LIN {X 0,Y 114.928,Z 408.229,A -85,B 0,C 180,E1 -30802.349,E2 -30802.349} C_VEL
LIN {X 0,Y 112.852,Z 415.99,A -85,B 0,C 180,E1 -30806.603,E2 -30806.603} C_VEL
LIN {X 0,Y 110.875,Z 424.848,A -85,B 0,C 180,E1 -30812.549,E2 -30812.549} C_VEL
LIN {X 0,Y 109.952,Z 432.134,A -85,B 0,C 180,E1 -30818.427,E2 -30818.427} C_VEL
LIN {X 0,Y 110.137,Z 438.588,A -85,B 0,C 180,E1 -30824.579,E2 -30824.579} C_VEL
LIN {X 0,Y 111.737,Z 444.355,A -85,B 0,C 180,E1 -30831.025,E2 -30831.025} C_VEL
LIN {X 0,Y 115.537,Z 449.975,A -85,B 0,C 180,E1 -30838.383,E2 -30838.383} C_VEL
LIN {X 0,Y 120.475,Z 454.059,A -85,B 0,C 180,E1 -30844.487,E2 -30844.487} C_VEL
LIN {X 0,Y 127.737,Z 457.673,A -85,B 0,C 180,E1 -30850.724,E2 -30850.724} C_VEL
LIN {X 0,Y 137.278,Z 460.508,A -85,B 0,C 180,E1 -30856.577,E2 -30856.577} C_VEL
LIN {X 0,Y 149.17,Z 462.456,A -85,B 0,C 180,E1 -30861.875,E2 -30861.875} C_VEL
LIN {X 0,Y 161.996,Z 463.408,A -85,B 0,C 180,E1 -30866.197,E2 -30866.197} C_VEL
LIN {X 0,Y 172.889,Z 463.546,A -85,B 0,C 180,E1 -30869.172,E2 -30869.172} C_VEL
LIN {X 0,Y 171.419,Z 463.614,A -85,B 0,C 180,E1 -30869.286,E2 -30869.286} C_VEL
LIN {X 0,Y 166.186,Z 463.751,A -85,B 0,C 180,E1 -30868.796,E2 -30868.796} C_VEL
LIN {X 0,Y 154.259,Z 463.825,A -85,B 0,C 180,E1 -30866.675,E2 -30866.675} C_VEL
LIN {X 0,Y 146.999,Z 463.619,A -85,B 0,C 180,E1 -30864.785,E2 -30864.785} C_VEL
LIN {X 0,Y 144.8,Z 463.468,A -85,B 0,C 180,E1 -30864.025,E2 -30864.025} C_VEL
LIN {X 0,Y 129.691,Z 461.525,A -85,B 0,C 180,E1 -30857.262,E2 -30857.262} C_VEL
LIN {X 0,Y 123.495,Z 460.082,A -85,B 0,C 180,E1 -30853.468,E2 -30853.468} C_VEL
LIN {X 0,Y 114.996,Z 456.746,A -85,B 0,C 180,E1 -30846.448,E2 -30846.448} C_VEL
LIN {X 0,Y 108.181,Z 451.593,A -85,B 0,C 180,E1 -30837.619,E2 -30837.619} C_VEL
LIN {X 0,Y 105.024,Z 446.619,A -85,B 0,C 180,E1 -30830.311,E2 -30830.311} C_VEL
LIN {X 0,Y 103.823,Z 441.564,A -85,B 0,C 180,E1 -30823.894,E2 -30823.894} C_VEL
LIN {X 0,Y 104.011,Z 435.561,A -85,B 0,C 180,E1 -30817.451,E2 -30817.451} C_VEL
LIN {X 0,Y 105.361,Z 428.686,A -85,B 0,C 180,E1 -30811.268,E2 -30811.268} C_VEL
LIN {X 0,Y 107.859,Z 420.234,A -85,B 0,C 180,E1 -30805.054,E2 -30805.054} C_VEL
LIN {X 0,Y 110.868,Z 411.549,A -85,B 0,C 180,E1 -30799.917,E2 -30799.917} C_VEL
LIN {X 0,Y 113.638,Z 403.688,A -85,B 0,C 180,E1 -30796.061,E2 -30796.061} C_VEL
LIN {X 0,Y 115.913,Z 396.746,A -85,B 0,C 180,E1 -30792.908,E2 -30792.908} C_VEL
LIN {X 0,Y 116.822,Z 392.502,A -85,B 0,C 180,E1 -30790.396,E2 -30790.396} C_VEL
LIN {X 0,Y 117.379,Z 389.446,A -85,B 0,C 180,E1 -30787.772,E2 -30787.772} C_VEL
LIN {X 0,Y 117.764,Z 386.797,A -85,B 0,C 180,E1 -30784.354,E2 -30784.354} C_VEL
LIN {X 0,Y 118.148,Z 384.921,A -85,B 0,C 180,E1 -30779.998,E2 -30779.998} C_VEL
LIN {X 0,Y 117.859,Z 385.788,A -85,B 0,C 180,E1 -30779.68,E2 -30779.68} C_VEL
LIN {X 0,Y 112.453,Z 398.556,A -85,B 0,C 180,E1 -30779.412,E2 -30779.412} C_VEL
LIN {X 0,Y 106.312,Z 409.458,A -85,B 0,C 180,E1 -30779.084,E2 -30779.084} C_VEL
LIN {X 0,Y 100.174,Z 418.396,A -85,B 0,C 180,E1 -30778.714,E2 -30778.714} C_VEL
LIN {X 0,Y 93.168,Z 426.917,A -85,B 0,C 180,E1 -30778.175,E2 -30778.175} C_VEL
LIN {X 0,Y 86.17,Z 434.129,A -85,B 0,C 180,E1 -30777.574,E2 -30777.574} C_VEL
LIN {X 0,Y 79.187,Z 440.326,A -85,B 0,C 180,E1 -30776.819,E2 -30776.819} C_VEL
LIN {X 0,Y 70.482,Z 446.858,A -85,B 0,C 180,E1 -30775.661,E2 -30775.661} C_VEL
LIN {X 0,Y 63.552,Z 451.36,A -85,B 0,C 180,E1 -30774.431,E2 -30774.431} C_VEL
LIN {X 0,Y 52.249,Z 457.3,A -85,B 0,C 180,E1 -30771.68,E2 -30771.68} C_VEL
LIN {X 0,Y 43.037,Z 461.18,A -85,B 0,C 180,E1 -30768.466,E2 -30768.466} C_VEL
LIN {X 0,Y 36.38,Z 463.552,A -85,B 0,C 180,E1 -30764.995,E2 -30764.995} C_VEL
LIN {X 0,Y 29.88,Z 465.354,A -85,B 0,C 180,E1 -30760.192,E2 -30760.192} C_VEL
LIN {X 0,Y 18.299,Z 467.822,A -85,B 0,C 180,E1 -30740.185,E2 -30740.185} C_VEL
LIN {X 0,Y 14.211,Z 468.422,A -85,B 0,C 180,E1 -30719.639,E2 -30719.639} C_VEL
LIN {X 0,Y 12.863,Z 468.588,A -85,B 0,C 180,E1 -30690,E2 -30690} C_VEL
LIN {X 0,Y 14.256,Z 468.423,A -85,B 0,C 180,E1 -30660.462,E2 -30660.462} C_VEL
LIN {X 0,Y 18.308,Z 467.822,A -85,B 0,C 180,E1 -30639.849,E2 -30639.849} C_VEL
LIN {X 0,Y 29.882,Z 465.355,A -85,B 0,C 180,E1 -30619.819,E2 -30619.819} C_VEL
LIN {X 0,Y 39.699,Z 462.4,A -85,B 0,C 180,E1 -30613.177,E2 -30613.177} C_VEL
LIN {X 0,Y 49.826,Z 458.409,A -85,B 0,C 180,E1 -30609.123,E2 -30609.123} C_VEL
LIN {X 0,Y 57.014,Z 455,A -85,B 0,C 180,E1 -30607.085,E2 -30607.085} C_VEL
LIN {X 0,Y 67.011,Z 449.169,A -85,B 0,C 180,E1 -30604.906,E2 -30604.906} C_VEL
LIN {X 0,Y 75.699,Z 443.075,A -85,B 0,C 180,E1 -30603.587,E2 -30603.587} C_VEL
LIN {X 0,Y 82.676,Z 437.38,A -85,B 0,C 180,E1 -30602.781,E2 -30602.781} C_VEL
LIN {X 0,Y 91.416,Z 428.834,A -85,B 0,C 180,E1 -30601.94,E2 -30601.94} C_VEL
LIN {X 0,Y 98.421,Z 420.663,A -85,B 0,C 180,E1 -30601.41,E2 -30601.41} C_VEL
LIN {X 0,Y 104.557,Z 412.158,A -85,B 0,C 180,E1 -30601.01,E2 -30601.01} C_VEL
LIN {X 0,Y 109.821,Z 403.45,A -85,B 0,C 180,E1 -30600.722,E2 -30600.722} C_VEL
LIN {X 0,Y 114.579,Z 393.859,A -85,B 0,C 180,E1 -30600.513,E2 -30600.513} C_VEL
LIN {X 0,Y 117.859,Z 385.789,A -85,B 0,C 180,E1 -30600.319,E2 -30600.319} C_VEL
LIN {X 0,Y 118.147,Z 384.922,A -85,B 0,C 180,E1 -30600.002,E2 -30600.002} C_VEL
LIN {X 0,Y 117.762,Z 386.791,A -85,B 0,C 180,E1 -30595.671,E2 -30595.671} C_VEL
LIN {X 0,Y 117.552,Z 388.558,A -85,B 0,C 180,E1 -30593.134,E2 -30593.134} C_VEL
LIN {X 0,Y 117.059,Z 391.295,A -85,B 0,C 180,E1 -30590.499,E2 -30590.499} C_VEL
LIN {X 0,Y 116.143,Z 395.768,A -85,B 0,C 180,E1 -30587.597,E2 -30587.597} C_VEL
LIN {X 0,Y 114.614,Z 400.732,A -85,B 0,C 180,E1 -30585.237,E2 -30585.237} C_VEL
LIN {X 0,Y 111.495,Z 409.774,A -85,B 0,C 180,E1 -30580.998,E2 -30580.998} C_VEL
LIN {X 0,Y 109.117,Z 416.554,A -85,B 0,C 180,E1 -30577.269,E2 -30577.269} C_VEL
LIN {X 0,Y 106.354,Z 425.079,A -85,B 0,C 180,E1 -30571.506,E2 -30571.506} C_VEL
LIN {X 0,Y 104.496,Z 432.383,A -85,B 0,C 180,E1 -30565.518,E2 -30565.518} C_VEL
LIN {X 0,Y 103.733,Z 438.549,A -85,B 0,C 180,E1 -30559.47,E2 -30559.47} C_VEL
LIN {X 0,Y 104.353,Z 444.734,A -85,B 0,C 180,E1 -30552.201,E2 -30552.201} C_VEL
LIN {X 0,Y 106.92,Z 450.051,A -85,B 0,C 180,E1 -30544.758,E2 -30544.758} C_VEL
LIN {X 0,Y 111.236,Z 454.337,A -85,B 0,C 180,E1 -30537.811,E2 -30537.811} C_VEL
LIN {X 0,Y 117.729,Z 457.962,A -85,B 0,C 180,E1 -30530.988,E2 -30530.988} C_VEL
LIN {X 0,Y 124.297,Z 460.268,A -85,B 0,C 180,E1 -30526.017,E2 -30526.017} C_VEL
LIN {X 0,Y 135.507,Z 462.502,A -85,B 0,C 180,E1 -30519.804,E2 -30519.804} C_VEL
LIN {X 0,Y 148.1,Z 463.65,A -85,B 0,C 180,E1 -30514.785,E2 -30514.785} C_VEL
LIN {X 0,Y 164.307,Z 463.8,A -85,B 0,C 180,E1 -30510,E2 -30510} C_VEL
LIN {X 0,Y 148.1,Z 463.65,A -85,B 0,C 180,E1 -30505.215,E2 -30505.215} C_VEL
LIN {X 0,Y 144.8,Z 463.468,A -85,B 0,C 180,E1 -30504.025,E2 -30504.025} C_VEL
LIN {X 0,Y 140.14,Z 463.214,A -85,B 0,C 180,E1 -30502.568,E2 -30502.568} C_VEL
LIN {X 0,Y 124.745,Z 462.622,A -85,B 0,C 180,E1 -30498.671,E2 -30498.671} C_VEL
LIN {X 0,Y 120.314,Z 462.099,A -85,B 0,C 180,E1 -30496.874,E2 -30496.874} C_VEL
LIN {X 0,Y 119.067,Z 461.847,A -85,B 0,C 180,E1 -30496.159,E2 -30496.159} C_VEL
LIN {X 0,Y 111.725,Z 459.856,A -85,B 0,C 180,E1 -30490.653,E2 -30490.653} C_VEL
LIN {X 0,Y 103.714,Z 455.76,A -85,B 0,C 180,E1 -30481.749,E2 -30481.749} C_VEL
LIN {X 0,Y 99.573,Z 451.39,A -85,B 0,C 180,E1 -30473.76,E2 -30473.76} C_VEL
LIN {X 0,Y 97.648,Z 446.43,A -85,B 0,C 180,E1 -30466.028,E2 -30466.028} C_VEL
LIN {X 0,Y 97.754,Z 439.952,A -85,B 0,C 180,E1 -30457.736,E2 -30457.736} C_VEL
LIN {X 0,Y 99.087,Z 434.239,A -85,B 0,C 180,E1 -30451.665,E2 -30451.665} C_VEL
LIN {X 0,Y 101.522,Z 427.548,A -85,B 0,C 180,E1 -30445.851,E2 -30445.851} C_VEL
LIN {X 0,Y 104.836,Z 419.615,A -85,B 0,C 180,E1 -30440.194,E2 -30440.194} C_VEL
LIN {X 0,Y 108.197,Z 411.955,A -85,B 0,C 180,E1 -30435.778,E2 -30435.778} C_VEL
LIN {X 0,Y 111.818,Z 403.365,A -85,B 0,C 180,E1 -30431.671,E2 -30431.671} C_VEL
LIN {X 0,Y 113.211,Z 399.616,A -85,B 0,C 180,E1 -30429.742,E2 -30429.742} C_VEL
LIN {X 0,Y 114.351,Z 395.944,A -85,B 0,C 180,E1 -30427.059,E2 -30427.059} C_VEL
LIN {X 0,Y 114.72,Z 394.322,A -85,B 0,C 180,E1 -30425.271,E2 -30425.271} C_VEL
LIN {X 0,Y 115.013,Z 393.127,A -85,B 0,C 180,E1 -30423.501,E2 -30423.501} C_VEL
LIN {X 0,Y 114.162,Z 394.978,A -85,B 0,C 180,E1 -30423.048,E2 -30423.048} C_VEL
LIN {X 0,Y 108.193,Z 406.5,A -85,B 0,C 180,E1 -30422.897,E2 -30422.897} C_VEL
LIN {X 0,Y 101.148,Z 417.069,A -85,B 0,C 180,E1 -30422.801,E2 -30422.801} C_VEL
LIN {X 0,Y 94.977,Z 424.806,A -85,B 0,C 180,E1 -30422.624,E2 -30422.624} C_VEL
LIN {X 0,Y 86.162,Z 433.936,A -85,B 0,C 180,E1 -30422.306,E2 -30422.306} C_VEL
LIN {X 0,Y 79.112,Z 440.133,A -85,B 0,C 180,E1 -30421.978,E2 -30421.978} C_VEL
LIN {X 0,Y 70.302,Z 446.665,A -85,B 0,C 180,E1 -30421.456,E2 -30421.456} C_VEL
LIN {X 0,Y 63.259,Z 451.165,A -85,B 0,C 180,E1 -30420.888,E2 -30420.888} C_VEL
LIN {X 0,Y 53.213,Z 456.436,A -85,B 0,C 180,E1 -30419.749,E2 -30419.749} C_VEL
LIN {X 0,Y 42.194,Z 460.986,A -85,B 0,C 180,E1 -30417.99,E2 -30417.99} C_VEL
LIN {X 0,Y 35.215,Z 463.358,A -85,B 0,C 180,E1 -30416.255,E2 -30416.255} C_VEL
LIN {X 0,Y 28.272,Z 465.161,A -85,B 0,C 180,E1 -30413.903,E2 -30413.903} C_VEL
LIN {X 0,Y 14.786,Z 467.628,A -85,B 0,C 180,E1 -30401.916,E2 -30401.916} C_VEL
LIN {X 0,Y 8.773,Z 468.229,A -85,B 0,C 180,E1 -30383.237,E2 -30383.237} C_VEL
LIN {X 0,Y 5.75,Z 468.395,A -85,B 0,C 180,E1 -30330,E2 -30330} C_VEL
LIN {X 0,Y 8.798,Z 468.23,A -85,B 0,C 180,E1 -30276.98,E2 -30276.98} C_VEL
LIN {X 0,Y 14.79,Z 467.629,A -85,B 0,C 180,E1 -30258.131,E2 -30258.131} C_VEL
LIN {X 0,Y 28.272,Z 465.161,A -85,B 0,C 180,E1 -30246.108,E2 -30246.108} C_VEL
LIN {X 0,Y 38.701,Z 462.206,A -85,B 0,C 180,E1 -30242.827,E2 -30242.827} C_VEL
LIN {X 0,Y 49.202,Z 458.215,A -85,B 0,C 180,E1 -30240.887,E2 -30240.887} C_VEL
LIN {X 0,Y 56.224,Z 455,A -85,B 0,C 180,E1 -30239.944,E2 -30239.944} C_VEL
LIN {X 0,Y 66.78,Z 448.975,A -85,B 0,C 180,E1 -30238.809,E2 -30238.809} C_VEL
LIN {X 0,Y 75.588,Z 442.882,A -85,B 0,C 180,E1 -30238.188,E2 -30238.188} C_VEL
LIN {X 0,Y 82.637,Z 437.187,A -85,B 0,C 180,E1 -30237.853,E2 -30237.853} C_VEL
LIN {X 0,Y 91.451,Z 428.641,A -85,B 0,C 180,E1 -30237.487,E2 -30237.487} C_VEL
LIN {X 0,Y 98.503,Z 420.47,A -85,B 0,C 180,E1 -30237.277,E2 -30237.277} C_VEL
LIN {X 0,Y 104.673,Z 411.965,A -85,B 0,C 180,E1 -30237.118,E2 -30237.118} C_VEL
LIN {X 0,Y 109.74,Z 403.667,A -85,B 0,C 180,E1 -30237.021,E2 -30237.021} C_VEL
LIN {X 0,Y 114.337,Z 394.575,A -85,B 0,C 180,E1 -30236.968,E2 -30236.968} C_VEL
LIN {X 0,Y 115.014,Z 393.125,A -85,B 0,C 180,E1 -30236.499,E2 -30236.499} C_VEL
LIN {X 0,Y 114.723,Z 394.314,A -85,B 0,C 180,E1 -30234.73,E2 -30234.73} C_VEL
LIN {X 0,Y 114.113,Z 396.916,A -85,B 0,C 180,E1 -30232.115,E2 -30232.115} C_VEL
LIN {X 0,Y 113.229,Z 399.587,A -85,B 0,C 180,E1 -30230.254,E2 -30230.254} C_VEL
LIN {X 0,Y 111.814,Z 403.367,A -85,B 0,C 180,E1 -30228.338,E2 -30228.338} C_VEL
LIN {X 0,Y 107.574,Z 413.501,A -85,B 0,C 180,E1 -30223.398,E2 -30223.398} C_VEL
LIN {X 0,Y 102.993,Z 423.981,A -85,B 0,C 180,E1 -30216.902,E2 -30216.902} C_VEL
LIN {X 0,Y 99.62,Z 432.673,A -85,B 0,C 180,E1 -30209.789,E2 -30209.789} C_VEL
LIN {X 0,Y 97.961,Z 438.801,A -85,B 0,C 180,E1 -30203.596,E2 -30203.596} C_VEL
LIN {X 0,Y 97.456,Z 444.881,A -85,B 0,C 180,E1 -30196.149,E2 -30196.149} C_VEL
LIN {X 0,Y 98.763,Z 450.06,A -85,B 0,C 180,E1 -30188.49,E2 -30188.49} C_VEL
LIN {X 0,Y 102.163,Z 454.476,A -85,B 0,C 180,E1 -30180.749,E2 -30180.749} C_VEL
LIN {X 0,Y 107.9,Z 458.25,A -85,B 0,C 180,E1 -30173.005,E2 -30173.005} C_VEL
LIN {X 0,Y 113.268,Z 460.373,A -85,B 0,C 180,E1 -30168.074,E2 -30168.074} C_VEL
LIN {X 0,Y 122.134,Z 462.489,A -85,B 0,C 180,E1 -30161.985,E2 -30161.985} C_VEL
LIN {X 0,Y 134.478,Z 463.878,A -85,B 0,C 180,E1 -30156,E2 -30156} C_VEL
LIN {X 0,Y 147.626,Z 464.245,A -85,B 0,C 180,E1 -30151.378,E2 -30151.378} C_VEL
LIN {X 0,Y 152.404,Z 464.117,A -85,B 0,C 180,E1 -30150,E2 -30150} C_VEL
LIN {X 0,Y 139.992,Z 464.098,A -85,B 0,C 180,E1 -30146.11,E2 -30146.11} C_VEL
LIN {X 0,Y 126.502,Z 463.069,A -85,B 0,C 180,E1 -30140.406,E2 -30140.406} C_VEL
LIN {X 0,Y 119.067,Z 461.847,A -85,B 0,C 180,E1 -30136.159,E2 -30136.159} C_VEL
LIN {X 0,Y 115.138,Z 461.181,A -85,B 0,C 180,E1 -30134.021,E2 -30134.021} C_VEL
LIN {X 0,Y 102.075,Z 459.573,A -85,B 0,C 180,E1 -30127.656,E2 -30127.656} C_VEL
LIN {X 0,Y 98.757,Z 458.636,A -85,B 0,C 180,E1 -30124.935,E2 -30124.935} C_VEL
LIN {X 0,Y 97.945,Z 458.238,A -85,B 0,C 180,E1 -30123.921,E2 -30123.921} C_VEL
LIN {X 0,Y 93.529,Z 454.579,A -85,B 0,C 180,E1 -30115.743,E2 -30115.743} C_VEL
LIN {X 0,Y 91.161,Z 449.41,A -85,B 0,C 180,E1 -30106.065,E2 -30106.065} C_VEL
LIN {X 0,Y 91.65,Z 442.9,A -85,B 0,C 180,E1 -30096.458,E2 -30096.458} C_VEL
LIN {X 0,Y 94.362,Z 435.211,A -85,B 0,C 180,E1 -30087.737,E2 -30087.737} C_VEL
LIN {X 0,Y 98.08,Z 427.571,A -85,B 0,C 180,E1 -30080.992,E2 -30080.992} C_VEL
LIN {X 0,Y 102.195,Z 419.847,A -85,B 0,C 180,E1 -30075.68,E2 -30075.68} C_VEL
LIN {X 0,Y 106.179,Z 412.266,A -85,B 0,C 180,E1 -30071.451,E2 -30071.451} C_VEL
LIN {X 0,Y 109.808,Z 404.92,A -85,B 0,C 180,E1 -30067.85,E2 -30067.85} C_VEL
LIN {X 0,Y 110.199,Z 403.982,A -85,B 0,C 180,E1 -30067.326,E2 -30067.326} C_VEL
LIN {X 0,Y 109.135,Z 405.681,A -85,B 0,C 180,E1 -30066.638,E2 -30066.638} C_VEL
LIN {X 0,Y 101.743,Z 416.876,A -85,B 0,C 180,E1 -30066.8,E2 -30066.8} C_VEL
LIN {X 0,Y 95.565,Z 424.614,A -85,B 0,C 180,E1 -30066.878,E2 -30066.878} C_VEL
LIN {X 0,Y 86.741,Z 433.743,A -85,B 0,C 180,E1 -30067.008,E2 -30067.008} C_VEL
LIN {X 0,Y 79.678,Z 439.939,A -85,B 0,C 180,E1 -30067.113,E2 -30067.113} C_VEL
LIN {X 0,Y 70.844,Z 446.471,A -85,B 0,C 180,E1 -30067.236,E2 -30067.236} C_VEL
LIN {X 0,Y 63.77,Z 450.972,A -85,B 0,C 180,E1 -30067.31,E2 -30067.31} C_VEL
LIN {X 0,Y 52.657,Z 456.683,A -85,B 0,C 180,E1 -30067.413,E2 -30067.413} C_VEL
LIN {X 0,Y 42.543,Z 460.793,A -85,B 0,C 180,E1 -30067.618,E2 -30067.618} C_VEL
LIN {X 0,Y 35.469,Z 463.165,A -85,B 0,C 180,E1 -30067.807,E2 -30067.807} C_VEL
LIN {X 0,Y 28.411,Z 464.968,A -85,B 0,C 180,E1 -30068.326,E2 -30068.326} C_VEL
LIN {X 0,Y 14.286,Z 467.434,A -85,B 0,C 180,E1 -30070.299,E2 -30070.299} C_VEL
LIN {X 0,Y 7.274,Z 468.036,A -85,B 0,C 180,E1 -30074.948,E2 -30074.948} C_VEL
LIN {X 0,Y 1.35,Z 468.202,A -85,B 0,C 180,E1 -30150,E2 -30150} C_VEL
LIN {X 0,Y 7.265,Z 468.037,A -85,B 0,C 180,E1 -30225.329,E2 -30225.329} C_VEL
LIN {X 0,Y 14.284,Z 467.435,A -85,B 0,C 180,E1 -30229.75,E2 -30229.75} C_VEL
LIN {X 0,Y 28.411,Z 464.968,A -85,B 0,C 180,E1 -30231.683,E2 -30231.683} C_VEL
LIN {X 0,Y 39.008,Z 462.012,A -85,B 0,C 180,E1 -30232.278,E2 -30232.278} C_VEL
LIN {X 0,Y 49.607,Z 458.021,A -85,B 0,C 180,E1 -30232.617,E2 -30232.617} C_VEL
LIN {X 0,Y 56.684,Z 454.805,A -85,B 0,C 180,E1 -30232.693,E2 -30232.693} C_VEL
LIN {X 0,Y 67.307,Z 448.782,A -85,B 0,C 180,E1 -30232.73,E2 -30232.73} C_VEL
LIN {X 0,Y 76.147,Z 442.688,A -85,B 0,C 180,E1 -30232.826,E2 -30232.826} C_VEL
LIN {X 0,Y 83.207,Z 436.994,A -85,B 0,C 180,E1 -30232.956,E2 -30232.956} C_VEL
LIN {X 0,Y 92.037,Z 428.448,A -85,B 0,C 180,E1 -30233.066,E2 -30233.066} C_VEL
LIN {X 0,Y 99.094,Z 420.277,A -85,B 0,C 180,E1 -30233.172,E2 -30233.172} C_VEL
LIN {X 0,Y 105.27,Z 411.772,A -85,B 0,C 180,E1 -30233.253,E2 -30233.253} C_VEL
LIN {X 0,Y 109.157,Z 405.655,A -85,B 0,C 180,E1 -30233.323,E2 -30233.323} C_VEL
LIN {X 0,Y 110.22,Z 403.943,A -85,B 0,C 180,E1 -30232.675,E2 -30232.675} C_VEL
LIN {X 0,Y 108.078,Z 408.522,A -85,B 0,C 180,E1 -30230.382,E2 -30230.382} C_VEL
LIN {X 0,Y 103.848,Z 416.786,A -85,B 0,C 180,E1 -30226.146,E2 -30226.146} C_VEL
LIN {X 0,Y 99.106,Z 425.626,A -85,B 0,C 180,E1 -30220.474,E2 -30220.474} C_VEL
LIN {X 0,Y 95.433,Z 432.915,A -85,B 0,C 180,E1 -30214.434,E2 -30214.434} C_VEL
LIN {X 0,Y 92.739,Z 439.22,A -85,B 0,C 180,E1 -30207.965,E2 -30207.965} C_VEL
LIN {X 0,Y 91.127,Z 445.139,A -85,B 0,C 180,E1 -30200.464,E2 -30200.464} C_VEL
LIN {X 0,Y 91.294,Z 450.224,A -85,B 0,C 180,E1 -30192.491,E2 -30192.491} C_VEL
LIN {X 0,Y 93.515,Z 454.591,A -85,B 0,C 180,E1 -30184.244,E2 -30184.244} C_VEL
LIN {X 0,Y 98.459,Z 458.531,A -85,B 0,C 180,E1 -30175.358,E2 -30175.358} C_VEL
LIN {X 0,Y 104.082,Z 460.928,A -85,B 0,C 180,E1 -30169.039,E2 -30169.039} C_VEL
LIN {X 0,Y 115.577,Z 463.37,A -85,B 0,C 180,E1 -30160.511,E2 -30160.511} C_VEL
LIN {X 0,Y 126.957,Z 464.345,A -85,B 0,C 180,E1 -30154.862,E2 -30154.862} C_VEL
LIN {X 0,Y 133.633,Z 464.588,A -85,B 0,C 180,E1 -30152.277,E2 -30152.277} C_VEL
LIN {X 0,Y 140.49,Z 464.434,A -85,B 0,C 180,E1 -30150,E2 -30150} C_VEL
LIN {X 0,Y 126.957,Z 464.344,A -85,B 0,C 180,E1 -30145.136,E2 -30145.136} C_VEL
LIN {X 0,Y 115.562,Z 463.37,A -85,B 0,C 180,E1 -30139.488,E2 -30139.488} C_VEL
LIN {X 0,Y 108.907,Z 462.223,A -85,B 0,C 180,E1 -30135.041,E2 -30135.041} C_VEL
LIN {X 0,Y 103.223,Z 460.661,A -85,B 0,C 180,E1 -30130.097,E2 -30130.097} C_VEL
LIN {X 0,Y 97.945,Z 458.238,A -85,B 0,C 180,E1 -30123.921,E2 -30123.921} C_VEL
LIN {X 0,Y 95.343,Z 457.153,A -85,B 0,C 180,E1 -30120.841,E2 -30120.841} C_VEL
LIN {X 0,Y 86.429,Z 454.259,A -85,B 0,C 180,E1 -30111.246,E2 -30111.246} C_VEL
LIN {X 0,Y 84.791,Z 452.786,A -85,B 0,C 180,E1 -30107.593,E2 -30107.593} C_VEL
LIN {X 0,Y 84.578,Z 452.165,A -85,B 0,C 180,E1 -30106.34,E2 -30106.34} C_VEL
LIN {X 0,Y 85.082,Z 446.716,A -85,B 0,C 180,E1 -30096.76,E2 -30096.76} C_VEL
LIN {X 0,Y 87.432,Z 440.989,A -85,B 0,C 180,E1 -30088.833,E2 -30088.833} C_VEL
LIN {X 0,Y 90.494,Z 435.565,A -85,B 0,C 180,E1 -30082.847,E2 -30082.847} C_VEL
LIN {X 0,Y 94.304,Z 429.452,A -85,B 0,C 180,E1 -30077.341,E2 -30077.341} C_VEL
LIN {X 0,Y 99.451,Z 421.347,A -85,B 0,C 180,E1 -30071.703,E2 -30071.703} C_VEL
LIN {X 0,Y 100.189,Z 420.084,A -85,B 0,C 180,E1 -30070.87,E2 -30070.87} C_VEL
LIN {X 0,Y 93.166,Z 428.254,A -85,B 0,C 180,E1 -30071.288,E2 -30071.288} C_VEL
LIN {X 0,Y 84.373,Z 436.801,A -85,B 0,C 180,E1 -30071.838,E2 -30071.838} C_VEL
LIN {X 0,Y 73.841,Z 445.123,A -85,B 0,C 180,E1 -30072.693,E2 -30072.693} C_VEL
LIN {X 0,Y 65.06,Z 450.779,A -85,B 0,C 180,E1 -30073.54,E2 -30073.54} C_VEL
LIN {X 0,Y 55.292,Z 455.933,A -85,B 0,C 180,E1 -30074.723,E2 -30074.723} C_VEL
LIN {X 0,Y 47.522,Z 459.36,A -85,B 0,C 180,E1 -30075.998,E2 -30075.998} C_VEL
LIN {X 0,Y 37.119,Z 462.971,A -85,B 0,C 180,E1 -30078.793,E2 -30078.793} C_VEL
LIN {X 0,Y 23.549,Z 466.17,A -85,B 0,C 180,E1 -30086.452,E2 -30086.452} C_VEL
LIN {X 0,Y 17.073,Z 467.241,A -85,B 0,C 180,E1 -30094.583,E2 -30094.583} C_VEL
LIN {X 0,Y 11.414,Z 467.843,A -85,B 0,C 180,E1 -30111.995,E2 -30111.995} C_VEL
LIN {X 0,Y 8.44,Z 468.01,A -85,B 0,C 180,E1 -30150,E2 -30150} C_VEL
LIN {X 0,Y 11.39,Z 467.843,A -85,B 0,C 180,E1 -30188.098,E2 -30188.098} C_VEL
LIN {X 0,Y 17.066,Z 467.241,A -85,B 0,C 180,E1 -30205.448,E2 -30205.448} C_VEL
LIN {X 0,Y 30.269,Z 464.775,A -85,B 0,C 180,E1 -30218.239,E2 -30218.239} C_VEL
LIN {X 0,Y 40.589,Z 461.818,A -85,B 0,C 180,E1 -30222.235,E2 -30222.235} C_VEL
LIN {X 0,Y 51.022,Z 457.827,A -85,B 0,C 180,E1 -30224.623,E2 -30224.623} C_VEL
LIN {X 0,Y 61.543,Z 452.695,A -85,B 0,C 180,E1 -30226.089,E2 -30226.089} C_VEL
LIN {X 0,Y 70.329,Z 447.433,A -85,B 0,C 180,E1 -30226.986,E2 -30226.986} C_VEL
LIN {X 0,Y 79.116,Z 441.12,A -85,B 0,C 180,E1 -30227.725,E2 -30227.725} C_VEL
LIN {X 0,Y 86.138,Z 435.175,A -85,B 0,C 180,E1 -30228.257,E2 -30228.257} C_VEL
LIN {X 0,Y 93.163,Z 428.255,A -85,B 0,C 180,E1 -30228.722,E2 -30228.722} C_VEL
LIN {X 0,Y 100.188,Z 420.084,A -85,B 0,C 180,E1 -30229.133,E2 -30229.133} C_VEL
LIN {X 0,Y 94.292,Z 429.466,A -85,B 0,C 180,E1 -30222.657,E2 -30222.657} C_VEL
LIN {X 0,Y 89.395,Z 437.538,A -85,B 0,C 180,E1 -30215.199,E2 -30215.199} C_VEL
LIN {X 0,Y 85.895,Z 444.537,A -85,B 0,C 180,E1 -30206.516,E2 -30206.516} C_VEL
LIN {X 0,Y 84.516,Z 449.745,A -85,B 0,C 180,E1 -30198.302,E2 -30198.302} C_VEL
LIN {X 0,Y 85.335,Z 454.643,A -85,B 0,C 180,E1 -30188.527,E2 -30188.527} C_VEL
LIN {X 0,Y 89.363,Z 458.807,A -85,B 0,C 180,E1 -30178.156,E2 -30178.156} C_VEL
LIN {X 0,Y 93.397,Z 460.947,A -85,B 0,C 180,E1 -30172.101,E2 -30172.101} C_VEL
LIN {X 0,Y 101.475,Z 463.156,A -85,B 0,C 180,E1 -30164.169,E2 -30164.169} C_VEL
LIN {X 0,Y 113.19,Z 464.541,A -85,B 0,C 180,E1 -30156.581,E2 -30156.581} C_VEL
LIN {X 0,Y 126.512,Z 464.807,A -85,B 0,C 180,E1 -30150.81,E2 -30150.81} C_VEL
LIN {X 0,Y 128.831,Z 464.745,A -85,B 0,C 180,E1 -30150,E2 -30150} C_VEL
LIN {X 0,Y 119.694,Z 464.822,A -85,B 0,C 180,E1 -30146.511,E2 -30146.511} C_VEL
LIN {X 0,Y 107.077,Z 463.976,A -85,B 0,C 180,E1 -30139.894,E2 -30139.894} C_VEL
LIN {X 0,Y 98.651,Z 462.513,A -85,B 0,C 180,E1 -30133.443,E2 -30133.443} C_VEL
LIN {X 0,Y 91.466,Z 460.037,A -85,B 0,C 180,E1 -30125.279,E2 -30125.279} C_VEL
LIN {X 0,Y 86.239,Z 455.94,A -85,B 0,C 180,E1 -30114.577,E2 -30114.577} C_VEL
LIN {X 0,Y 84.578,Z 452.165,A -85,B 0,C 180,E1 -30106.34,E2 -30106.34} C_VEL
LIN {X 0,Y 83.854,Z 450.444,A -85,B 0,C 180,E1 -30102.514,E2 -30102.514} C_VEL
LIN {X 0,Y 81.236,Z 446.018,A -85,B 0,C 180,E1 -30090.633,E2 -30090.633} C_VEL
LIN {X 0,Y 81.794,Z 443.901,A -85,B 0,C 180,E1 -30086.8,E2 -30086.8} C_VEL
LIN {X 0,Y 82.275,Z 443.038,A -85,B 0,C 180,E1 -30085.617,E2 -30085.617} C_VEL
LIN {X 0,Y 87.313,Z 435.949,A -85,B 0,C 180,E1 -30077.577,E2 -30077.577} C_VEL
LIN {X 0,Y 88.021,Z 434.966,A -85,B 0,C 180,E1 -30076.639,E2 -30076.639} C_VEL
LIN {X 0,Y 87.863,Z 434.982,A -85,B 0,C 180,E1 -30076.29,E2 -30076.29} C_VEL
LIN {X 0,Y 80.923,Z 440.927,A -85,B 0,C 180,E1 -30077.191,E2 -30077.191} C_VEL
LIN {X 0,Y 72.272,Z 447.24,A -85,B 0,C 180,E1 -30078.536,E2 -30078.536} C_VEL
LIN {X 0,Y 63.641,Z 452.501,A -85,B 0,C 180,E1 -30080.17,E2 -30080.17} C_VEL
LIN {X 0,Y 53.369,Z 457.633,A -85,B 0,C 180,E1 -30082.809,E2 -30082.809} C_VEL
LIN {X 0,Y 43.304,Z 461.624,A -85,B 0,C 180,E1 -30086.796,E2 -30086.796} C_VEL
LIN {X 0,Y 33.563,Z 464.582,A -85,B 0,C 180,E1 -30093.115,E2 -30093.115} C_VEL
LIN {X 0,Y 21.919,Z 467.047,A -85,B 0,C 180,E1 -30110.113,E2 -30110.113} C_VEL
LIN {X 0,Y 17.57,Z 467.65,A -85,B 0,C 180,E1 -30126.422,E2 -30126.422} C_VEL
LIN {X 0,Y 15.549,Z 467.817,A -85,B 0,C 180,E1 -30150,E2 -30150} C_VEL
LIN {X 0,Y 17.547,Z 467.65,A -85,B 0,C 180,E1 -30173.611,E2 -30173.611} C_VEL
LIN {X 0,Y 21.911,Z 467.047,A -85,B 0,C 180,E1 -30189.904,E2 -30189.904} C_VEL
LIN {X 0,Y 33.561,Z 464.582,A -85,B 0,C 180,E1 -30206.891,E2 -30206.891} C_VEL
LIN {X 0,Y 43.302,Z 461.624,A -85,B 0,C 180,E1 -30213.208,E2 -30213.208} C_VEL
LIN {X 0,Y 53.361,Z 457.633,A -85,B 0,C 180,E1 -30217.211,E2 -30217.211} C_VEL
LIN {X 0,Y 63.639,Z 452.501,A -85,B 0,C 180,E1 -30219.833,E2 -30219.833} C_VEL
LIN {X 0,Y 72.272,Z 447.24,A -85,B 0,C 180,E1 -30221.464,E2 -30221.464} C_VEL
LIN {X 0,Y 80.927,Z 440.927,A -85,B 0,C 180,E1 -30222.801,E2 -30222.801} C_VEL
LIN {X 0,Y 87.865,Z 434.982,A -85,B 0,C 180,E1 -30223.706,E2 -30223.706} C_VEL
LIN {X 0,Y 88.035,Z 434.965,A -85,B 0,C 180,E1 -30223.332,E2 -30223.332} C_VEL
LIN {X 0,Y 83.132,Z 441.707,A -85,B 0,C 180,E1 -30216.033,E2 -30216.033} C_VEL
LIN {X 0,Y 79.399,Z 448.009,A -85,B 0,C 180,E1 -30206.882,E2 -30206.882} C_VEL
LIN {X 0,Y 77.855,Z 453.539,A -85,B 0,C 180,E1 -30196.233,E2 -30196.233} C_VEL
LIN {X 0,Y 78.947,Z 457.333,A -85,B 0,C 180,E1 -30186.76,E2 -30186.76} C_VEL
LIN {X 0,Y 84.529,Z 461.439,A -85,B 0,C 180,E1 -30173.862,E2 -30173.862} C_VEL
LIN {X 0,Y 88.798,Z 462.868,A -85,B 0,C 180,E1 -30168.249,E2 -30168.249} C_VEL
LIN {X 0,Y 101.15,Z 464.784,A -85,B 0,C 180,E1 -30157.988,E2 -30157.988} C_VEL
LIN {X 0,Y 112.511,Z 465.186,A -85,B 0,C 180,E1 -30151.979,E2 -30151.979} C_VEL
LIN {X 0,Y 117.267,Z 465.056,A -85,B 0,C 180,E1 -30150,E2 -30150} C_VEL
LIN {X 0,Y 105.856,Z 465.008,A -85,B 0,C 180,E1 -30144.771,E2 -30144.771} C_VEL
LIN {X 0,Y 99.607,Z 464.689,A -85,B 0,C 180,E1 -30141.027,E2 -30141.027} C_VEL
LIN {X 0,Y 88.582,Z 462.799,A -85,B 0,C 180,E1 -30131.497,E2 -30131.497} C_VEL
LIN {X 0,Y 84.016,Z 461.224,A -85,B 0,C 180,E1 -30125.276,E2 -30125.276} C_VEL
LIN {X 0,Y 78.993,Z 457.3,A -85,B 0,C 180,E1 -30113.195,E2 -30113.195} C_VEL
LIN {X 0,Y 77.866,Z 453.539,A -85,B 0,C 180,E1 -30103.776,E2 -30103.776} C_VEL
LIN {X 0,Y 79.262,Z 448.291,A -85,B 0,C 180,E1 -30093.558,E2 -30093.558} C_VEL
LIN {X 0,Y 82.275,Z 443.038,A -85,B 0,C 180,E1 -30085.617,E2 -30085.617} C_VEL
LIN {X 0,Y 81.943,Z 442.977,A -85,B 0,C 180,E1 -30084.911,E2 -30084.911} C_VEL
LIN {X 0,Y 80.234,Z 443.849,A -85,B 0,C 180,E1 -30084.111,E2 -30084.111} C_VEL
LIN {X 0,Y 76.621,Z 445.988,A -85,B 0,C 180,E1 -30083.791,E2 -30083.791} C_VEL
LIN {X 0,Y 70.009,Z 450.277,A -85,B 0,C 180,E1 -30084.983,E2 -30084.983} C_VEL
LIN {X 0,Y 63.924,Z 453.75,A -85,B 0,C 180,E1 -30086.731,E2 -30086.731} C_VEL
LIN {X 0,Y 53.26,Z 458.972,A -85,B 0,C 180,E1 -30090.939,E2 -30090.939} C_VEL
LIN {X 0,Y 43.866,Z 462.583,A -85,B 0,C 180,E1 -30096.767,E2 -30096.767} C_VEL
LIN {X 0,Y 37.938,Z 464.388,A -85,B 0,C 180,E1 -30102.183,E2 -30102.183} C_VEL
LIN {X 0,Y 27.761,Z 466.854,A -85,B 0,C 180,E1 -30119.581,E2 -30119.581} C_VEL
LIN {X 0,Y 24.275,Z 467.456,A -85,B 0,C 180,E1 -30133.171,E2 -30133.171} C_VEL
LIN {X 0,Y 22.647,Z 467.624,A -85,B 0,C 180,E1 -30150,E2 -30150} C_VEL
LIN {X 0,Y 24.255,Z 467.457,A -85,B 0,C 180,E1 -30166.843,E2 -30166.843} C_VEL
LIN {X 0,Y 27.753,Z 466.854,A -85,B 0,C 180,E1 -30180.429,E2 -30180.429} C_VEL
LIN {X 0,Y 37.935,Z 464.388,A -85,B 0,C 180,E1 -30197.821,E2 -30197.821} C_VEL
LIN {X 0,Y 46.947,Z 461.431,A -85,B 0,C 180,E1 -30205.422,E2 -30205.422} C_VEL
LIN {X 0,Y 56.508,Z 457.44,A -85,B 0,C 180,E1 -30210.528,E2 -30210.528} C_VEL
LIN {X 0,Y 66.438,Z 452.307,A -85,B 0,C 180,E1 -30214.046,E2 -30214.046} C_VEL
LIN {X 0,Y 74.839,Z 447.046,A -85,B 0,C 180,E1 -30216.292,E2 -30216.292} C_VEL
LIN {X 0,Y 76.575,Z 445.888,A -85,B 0,C 180,E1 -30216.606,E2 -30216.606} C_VEL
LIN {X 0,Y 72.481,Z 451.702,A -85,B 0,C 180,E1 -30206.294,E2 -30206.294} C_VEL
LIN {X 0,Y 71.127,Z 455.902,A -85,B 0,C 180,E1 -30196.243,E2 -30196.243} C_VEL
LIN {X 0,Y 72.261,Z 459.353,A -85,B 0,C 180,E1 -30185.701,E2 -30185.701} C_VEL
LIN {X 0,Y 74.897,Z 461.5,A -85,B 0,C 180,E1 -30177.981,E2 -30177.981} C_VEL
LIN {X 0,Y 81.174,Z 463.741,A -85,B 0,C 180,E1 -30167.764,E2 -30167.764} C_VEL
LIN {X 0,Y 92.19,Z 465.166,A -85,B 0,C 180,E1 -30157.695,E2 -30157.695} C_VEL
LIN {X 0,Y 98.592,Z 465.473,A -85,B 0,C 180,E1 -30153.683,E2 -30153.683} C_VEL
LIN {X 0,Y 105.989,Z 465.362,A -85,B 0,C 180,E1 -30150,E2 -30150} C_VEL
LIN {X 0,Y 97.797,Z 465.439,A -85,B 0,C 180,E1 -30145.879,E2 -30145.879} C_VEL
LIN {X 0,Y 86.329,Z 464.603,A -85,B 0,C 180,E1 -30137.651,E2 -30137.651} C_VEL
LIN {X 0,Y 78.859,Z 463.079,A -85,B 0,C 180,E1 -30129.116,E2 -30129.116} C_VEL
LIN {X 0,Y 73.735,Z 460.696,A -85,B 0,C 180,E1 -30119.068,E2 -30119.068} C_VEL
LIN {X 0,Y 71.162,Z 456.799,A -85,B 0,C 180,E1 -30106.265,E2 -30106.265} C_VEL
LIN {X 0,Y 71.991,Z 452.703,A -85,B 0,C 180,E1 -30095.851,E2 -30095.851} C_VEL
LIN {X 0,Y 74.87,Z 448.093,A -85,B 0,C 180,E1 -30086.906,E2 -30086.906} C_VEL
LIN {X 0,Y 76.522,Z 445.892,A -85,B 0,C 180,E1 -30083.303,E2 -30083.303} C_VEL
LIN {X 0,Y 69.791,Z 450.391,A -85,B 0,C 180,E1 -30085.001,E2 -30085.001} C_VEL
LIN {X 0,Y 63.924,Z 453.75,A -85,B 0,C 180,E1 -30086.731,E2 -30086.731} C_VEL
LIN {X 0,Y 59.269,Z 456.419,A -85,B 0,C 180,E1 -30089.052,E2 -30089.052} C_VEL
LIN {X 0,Y 52.616,Z 460.127,A -85,B 0,C 180,E1 -30095.592,E2 -30095.592} C_VEL
LIN {X 0,Y 46.63,Z 462.971,A -85,B 0,C 180,E1 -30104.174,E2 -30104.174} C_VEL
LIN {X 0,Y 42.731,Z 464.283,A -85,B 0,C 180,E1 -30109.648,E2 -30109.648} C_VEL
LIN {X 0,Y 34.106,Z 466.66,A -85,B 0,C 180,E1 -30125.661,E2 -30125.661} C_VEL
LIN {X 0,Y 31.16,Z 467.263,A -85,B 0,C 180,E1 -30136.965,E2 -30136.965} C_VEL
LIN {X 0,Y 29.762,Z 467.431,A -85,B 0,C 180,E1 -30150,E2 -30150} C_VEL
LIN {X 0,Y 31.142,Z 467.263,A -85,B 0,C 180,E1 -30163.042,E2 -30163.042} C_VEL
LIN {X 0,Y 34.098,Z 466.66,A -85,B 0,C 180,E1 -30174.345,E2 -30174.345} C_VEL
LIN {X 0,Y 43.052,Z 464.194,A -85,B 0,C 180,E1 -30190.766,E2 -30190.766} C_VEL
LIN {X 0,Y 51.323,Z 461.237,A -85,B 0,C 180,E1 -30198.864,E2 -30198.864} C_VEL
LIN {X 0,Y 60.344,Z 457.246,A -85,B 0,C 180,E1 -30204.613,E2 -30204.613} C_VEL
LIN {X 0,Y 61.831,Z 456.502,A -85,B 0,C 180,E1 -30205.371,E2 -30205.371} C_VEL
LIN {X 0,Y 65.575,Z 454.966,A -85,B 0,C 180,E1 -30205.855,E2 -30205.855} C_VEL
LIN {X 0,Y 64.35,Z 458.554,A -85,B 0,C 180,E1 -30194.983,E2 -30194.983} C_VEL
LIN {X 0,Y 66.247,Z 461.795,A -85,B 0,C 180,E1 -30181.936,E2 -30181.936} C_VEL
LIN {X 0,Y 73.553,Z 464.442,A -85,B 0,C 180,E1 -30167.169,E2 -30167.169} C_VEL
LIN {X 0,Y 79.974,Z 465.366,A -85,B 0,C 180,E1 -30160.123,E2 -30160.123} C_VEL
LIN {X 0,Y 91.41,Z 465.759,A -85,B 0,C 180,E1 -30151.893,E2 -30151.893} C_VEL
LIN {X 0,Y 94.915,Z 465.662,A -85,B 0,C 180,E1 -30150,E2 -30150} C_VEL
LIN {X 0,Y 84.814,Z 465.631,A -85,B 0,C 180,E1 -30143.886,E2 -30143.886} C_VEL
LIN {X 0,Y 78.807,Z 465.287,A -85,B 0,C 180,E1 -30138.792,E2 -30138.792} C_VEL
LIN {X 0,Y 69.302,Z 463.308,A -85,B 0,C 180,E1 -30125.874,E2 -30125.874} C_VEL
LIN {X 0,Y 65.254,Z 460.777,A -85,B 0,C 180,E1 -30113.843,E2 -30113.843} C_VEL
LIN {X 0,Y 64.361,Z 458.555,A -85,B 0,C 180,E1 -30105.03,E2 -30105.03} C_VEL
LIN {X 0,Y 65.589,Z 454.96,A -85,B 0,C 180,E1 -30094.145,E2 -30094.145} C_VEL
LIN {X 0,Y 61.601,Z 456.625,A -85,B 0,C 180,E1 -30094.777,E2 -30094.777} C_VEL
LIN {X 0,Y 54.232,Z 460.02,A -85,B 0,C 180,E1 -30098.963,E2 -30098.963} C_VEL
LIN {X 0,Y 48.48,Z 462.389,A -85,B 0,C 180,E1 -30103.545,E2 -30103.545} C_VEL
LIN {X 0,Y 42.731,Z 464.283,A -85,B 0,C 180,E1 -30109.648,E2 -30109.648} C_VEL
LIN {X 0,Y 39.191,Z 465.457,A -85,B 0,C 180,E1 -30116.111,E2 -30116.111} C_VEL
LIN {X 0,Y 36.992,Z 466.387,A -85,B 0,C 180,E1 -30124.311,E2 -30124.311} C_VEL
LIN {X 0,Y 36.188,Z 467.263,A -85,B 0,C 180,E1 -30143.017,E2 -30143.017} C_VEL
LIN {X 0,Y 37.32,Z 467.155,A -85,B 0,C 180,E1 -30155.343,E2 -30155.343} C_VEL
LIN {X 0,Y 40.698,Z 466.467,A -85,B 0,C 180,E1 -30170.204,E2 -30170.204} C_VEL
LIN {X 0,Y 48.675,Z 464.001,A -85,B 0,C 180,E1 -30185.278,E2 -30185.278} C_VEL
LIN {X 0,Y 53.644,Z 462.196,A -85,B 0,C 180,E1 -30190.924,E2 -30190.924} C_VEL
LIN {X 0,Y 57.545,Z 460.835,A -85,B 0,C 180,E1 -30192.886,E2 -30192.886} C_VEL
LIN {X 0,Y 60.36,Z 463.63,A -85,B 0,C 180,E1 -30177.758,E2 -30177.758} C_VEL
LIN {X 0,Y 69.642,Z 465.652,A -85,B 0,C 180,E1 -30161.644,E2 -30161.644} C_VEL
LIN {X 0,Y 77.526,Z 466.082,A -85,B 0,C 180,E1 -30154.341,E2 -30154.341} C_VEL
LIN {X 0,Y 83.963,Z 465.96,A -85,B 0,C 180,E1 -30150,E2 -30150} C_VEL
LIN {X 0,Y 76.292,Z 466.025,A -85,B 0,C 180,E1 -30144.714,E2 -30144.714} C_VEL
LIN {X 0,Y 65.954,Z 465.137,A -85,B 0,C 180,E1 -30133.532,E2 -30133.532} C_VEL
LIN {X 0,Y 60.395,Z 463.628,A -85,B 0,C 180,E1 -30122.26,E2 -30122.26} C_VEL
LIN {X 0,Y 57.56,Z 460.827,A -85,B 0,C 180,E1 -30107.099,E2 -30107.099} C_VEL
LIN {X 0,Y 53.646,Z 462.195,A -85,B 0,C 180,E1 -30109.078,E2 -30109.078} C_VEL
LIN {X 0,Y 47.915,Z 464.232,A -85,B 0,C 180,E1 -30115.783,E2 -30115.783} C_VEL
LIN {X 0,Y 40.725,Z 466.466,A -85,B 0,C 180,E1 -30129.81,E2 -30129.81} C_VEL
LIN {X 0,Y 38.124,Z 467.07,A -85,B 0,C 180,E1 -30139.377,E2 -30139.377} C_VEL
LIN {X 0,Y 36.867,Z 467.238,A -85,B 0,C 180,E1 -30150,E2 -30150} C_VEL
LIN {X 0,Y 37.32,Z 467.155,A -85,B 0,C 180,E1 -30155.343,E2 -30155.343} C_VEL
LIN {X 0,Y 38.707,Z 467.037,A -85,B 0,C 180,E1 -30160.913,E2 -30160.913} C_VEL
LIN {X 0,Y 43.06,Z 466.459,A -85,B 0,C 180,E1 -30167.901,E2 -30167.901} C_VEL
LIN {X 0,Y 51.868,Z 464.975,A -85,B 0,C 180,E1 -30175.508,E2 -30175.508} C_VEL
LIN {X 0,Y 53.35,Z 464.681,A -85,B 0,C 180,E1 -30176.679,E2 -30176.679} C_VEL
LIN {X 0,Y 59.614,Z 465.931,A -85,B 0,C 180,E1 -30163.638,E2 -30163.638} C_VEL
LIN {X 0,Y 70.325,Z 466.331,A -85,B 0,C 180,E1 -30152.146,E2 -30152.146} C_VEL
LIN {X 0,Y 73.206,Z 466.252,A -85,B 0,C 180,E1 -30150,E2 -30150} C_VEL
LIN {X 0,Y 63.886,Z 466.205,A -85,B 0,C 180,E1 -30141.893,E2 -30141.893} C_VEL
LIN {X 0,Y 58.377,Z 465.81,A -85,B 0,C 180,E1 -30134.377,E2 -30134.377} C_VEL
LIN {X 0,Y 53.369,Z 464.675,A -85,B 0,C 180,E1 -30123.288,E2 -30123.288} C_VEL
LIN {X 0,Y 50.742,Z 465.202,A -85,B 0,C 180,E1 -30125.449,E2 -30125.449} C_VEL
LIN {X 0,Y 47.496,Z 466.272,A -85,B 0,C 180,E1 -30132.786,E2 -30132.786} C_VEL
LIN {X 0,Y 45.147,Z 466.876,A -85,B 0,C 180,E1 -30141.044,E2 -30141.044} C_VEL
LIN {X 0,Y 43.963,Z 467.046,A -85,B 0,C 180,E1 -30150,E2 -30150} C_VEL
LIN {X 0,Y 45.115,Z 466.877,A -85,B 0,C 180,E1 -30158.962,E2 -30158.962} C_VEL
LIN {X 0,Y 47.47,Z 466.273,A -85,B 0,C 180,E1 -30167.223,E2 -30167.223} C_VEL
LIN {X 0,Y 50.736,Z 465.202,A -85,B 0,C 180,E1 -30174.555,E2 -30174.555} C_VEL
LIN {X 0,Y 51.868,Z 464.975,A -85,B 0,C 180,E1 -30175.508,E2 -30175.508} C_VEL
LIN {X 0,Y 52.759,Z 464.923,A -85,B 0,C 180,E1 -30175.309,E2 -30175.309} C_VEL
LIN {X 0,Y 53.81,Z 465.083,A -85,B 0,C 180,E1 -30173.499,E2 -30173.499} C_VEL
LIN {X 0,Y 54.545,Z 465.659,A -85,B 0,C 180,E1 -30168.656,E2 -30168.656} C_VEL
LIN {X 0,Y 55.549,Z 466.484,A -85,B 0,C 180,E1 -30159.057,E2 -30159.057} C_VEL
LIN {X 0,Y 57.558,Z 466.67,A -85,B 0,C 180,E1 -30154.933,E2 -30154.933} C_VEL
LIN {X 0,Y 58.144,Z 466.619,A -85,B 0,C 180,E1 -30154.246,E2 -30154.246} C_VEL
LIN {X 0,Y 62.625,Z 466.539,A -85,B 0,C 180,E1 -30150,E2 -30150} C_VEL
LIN {X 0,Y 54.097,Z 466.505,A -85,B 0,C 180,E1 -30140.837,E2 -30140.837} C_VEL
LIN {X 0,Y 52.212,Z 466.682,A -85,B 0,C 180,E1 -30142.264,E2 -30142.264} C_VEL
LIN {X 0,Y 51.086,Z 466.852,A -85,B 0,C 180,E1 -30150,E2 -30150} C_VEL
LIN {X 0,Y 52.181,Z 466.683,A -85,B 0,C 180,E1 -30157.74,E2 -30157.74} C_VEL
LIN {X 0,Y 54.083,Z 466.505,A -85,B 0,C 180,E1 -30159.18,E2 -30159.18} C_VEL
LIN {X 0,Y 58.144,Z 466.619,A -85,B 0,C 180,E1 -30154.246,E2 -30154.246} C_VEL
LIN {X 0,Y 59.541,Z 468.619,A -85,B 0,C 180,E1 -30152.818,E2 -30152.818} C_VEL
LIN {X 0,Y 59.541,Z 600,A -85,B 0,C 180,E1 -30152.818,E2 -30152.818} C_VEL
LIN {X 0,Y 59.541,Z 600,A -85,B 0,C 180,E1 -30152.818,E2 -30152.818}

QRS_NEXT_CUT()

QRS_NEXT()
QRS_HOME()

END
